SUBAPPLICATION AuxInput_Auseinanderklappen (* Subapplication Type *)
  (* Standard: 61499-2 *)
  (* Version 1.0, 2023-02-11, franz *)
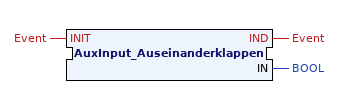
  EVENT_INPUT
    INIT;
  END_EVENT
  EVENT_OUTPUT
    IND;
  END_EVENT
  VAR_OUTPUT
    IN : BOOL;
  END_VAR
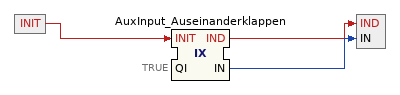
  FBS
    AuxInput_Auseinanderklappen : IX(QI := TRUE);
  END_FBS
  EVENT_CONNECTIONS
    INIT TO AuxInput_Auseinanderklappen.INIT;
    AuxInput_Auseinanderklappen.IND TO IND;
  END_CONNECTIONS
  DATA_CONNECTIONS
    AuxInput_Auseinanderklappen.IN TO IN;
  END_CONNECTIONS
END_SUBAPPLICATION
